Staubli VAL3: EditMain.pgx

public program EditMain(string x_sPath)
  local num l_nKey
  local bool l_bRes
begin
  //

  //
  //load path

    call loadPath(l_bRes,x_sPath)
    if !l_bRes
      return
    endIf

    //
    bUserRefresh=bListRefresh=true
    nPage=1
    //
    do
      call Refresh1()
      call RefreshList()
      call user:setList(x_sPath,sList,bUserRefresh,bListRefresh,nSelected,sItem,l_nKey)
      bUserRefresh=false
      bListRefresh=false
      call MainKey(l_nKey)
      delay(0)
    until bExit
    nPage=0
    bExit=false
    bUserRefresh=bListRefresh=true

end
